// TIA Portal V20 export
TYPE "s_PLC_Interlocks"
// stored: Access Published, IsFailsafeCompliant true, Namespace Safety
   STRUCT
      "Connection status" : "Safety.s_CONNECTION_STATUS";
      CellInterlocks : "Safety.s_zc_CellInterlocks";
      InterlockToAdjCellICSD : "Safety.s_zc_IntercellSafetyDeviceToAdjCell";
      NormalInterlocks : "Safety.s_zc_NormalInterlocks";
      MiscInterlock : "Safety.s_zc_MiscInterlocks";
   END_STRUCT;
   // // NormalInterlocks.reserved02 : BA60 JR PP Left Door Open (Stack#1)
   // // NormalInterlocks.reserved03 : BA60 Top Tape Door Open (Stack#2)
   // // NormalInterlocks.reserved04 : BA60 JR PP Left Door Forced Open (Stackr#1)
   // // NormalInterlocks.reserved05 : BA60 Top Tape Door Forced Open (Stackr#2)
   // // NormalInterlocks.reserved06 : BA60 External Door Open (Stackr#1)
   // // NormalInterlocks.reserved07 : BA60 External Door Open (Stackr#2)
   // // NormalInterlocks.reserved08 : Cathode Conveyor Cover Closed
   // // NormalInterlocks.reserved09 : Anode Conveyor Cover Closed
   // // NormalInterlocks.reserved10 : BA60 Light Curtain Muting (Stack#1)
   // // NormalInterlocks.reserved11 : BA60 Light Curtain NOK (Stack#1)
   // // NormalInterlocks.reserved12 : BA60 Light Curtain Muting (Stack#2)
   // // NormalInterlocks.reserved13 : BA60 Light Curtain NOK (Stack#2)
END_TYPE
